# EPICS autosave request: ADApp/Db/CCDMultiTrack_settings.req
$(P)$(R)CCDMultiTrackStart
$(P)$(R)CCDMultiTrackEnd
$(P)$(R)CCDMultiTrackBin
